// TIA Portal V17 export
// export: Created 2025-07-01T09:58:25.2131058Z, ExportSetting WithDefaults, DisplayName Totally Integrated Automation Portal, DisplayVersion V17 Update 8, DisplayName TIA Portal Openness, DisplayVersion V17 Update 8, DisplayName TIA Portal Version Control Interface, DisplayVersion V17, DisplayName SINAMICS Startdrive Advanced, DisplayVersion V17 SP2, DisplayName SINAMICS Startdrive G110M, G120, G120C, G120D, G120P, G115D, DisplayVersion V17 SP2, DisplayName SINAMICS Startdrive G130, G150, S120, S150, SINAMICS MV, S210, DisplayVersion V17 SP2, DisplayName STEP 7 Professional, DisplayVersion V17 Update 8, DisplayName SINUMERIK ONE STEP 7 Toolbox, DisplayVersion V17 Update 12, DisplayName SINUMERIK ONE PLC Basic Program Plus, DisplayVersion V17 Update 12, DisplayName SINUMERIK 840D sl STEP 7 Toolbox, DisplayVersion V17 Update 12, DisplayName STEP 7 Safety, DisplayVersion V17 Update 6, DisplayName WinCC Advanced, DisplayVersion V17 Update 8
FUNCTION "FC2441_MACHINE_STATUS" : Void   // FC2441, LAD
{ S7_Optimized_Access := 'TRUE' }
VERSION : 0.1
// stored: AutoNumber false, IsIECCheckEnabled false, SetENOAutomatically false, UDAEnableTagReadback false
BEGIN

REGION Network 1: UNIT 1 STATION 3 CLADDING IN PROCESS
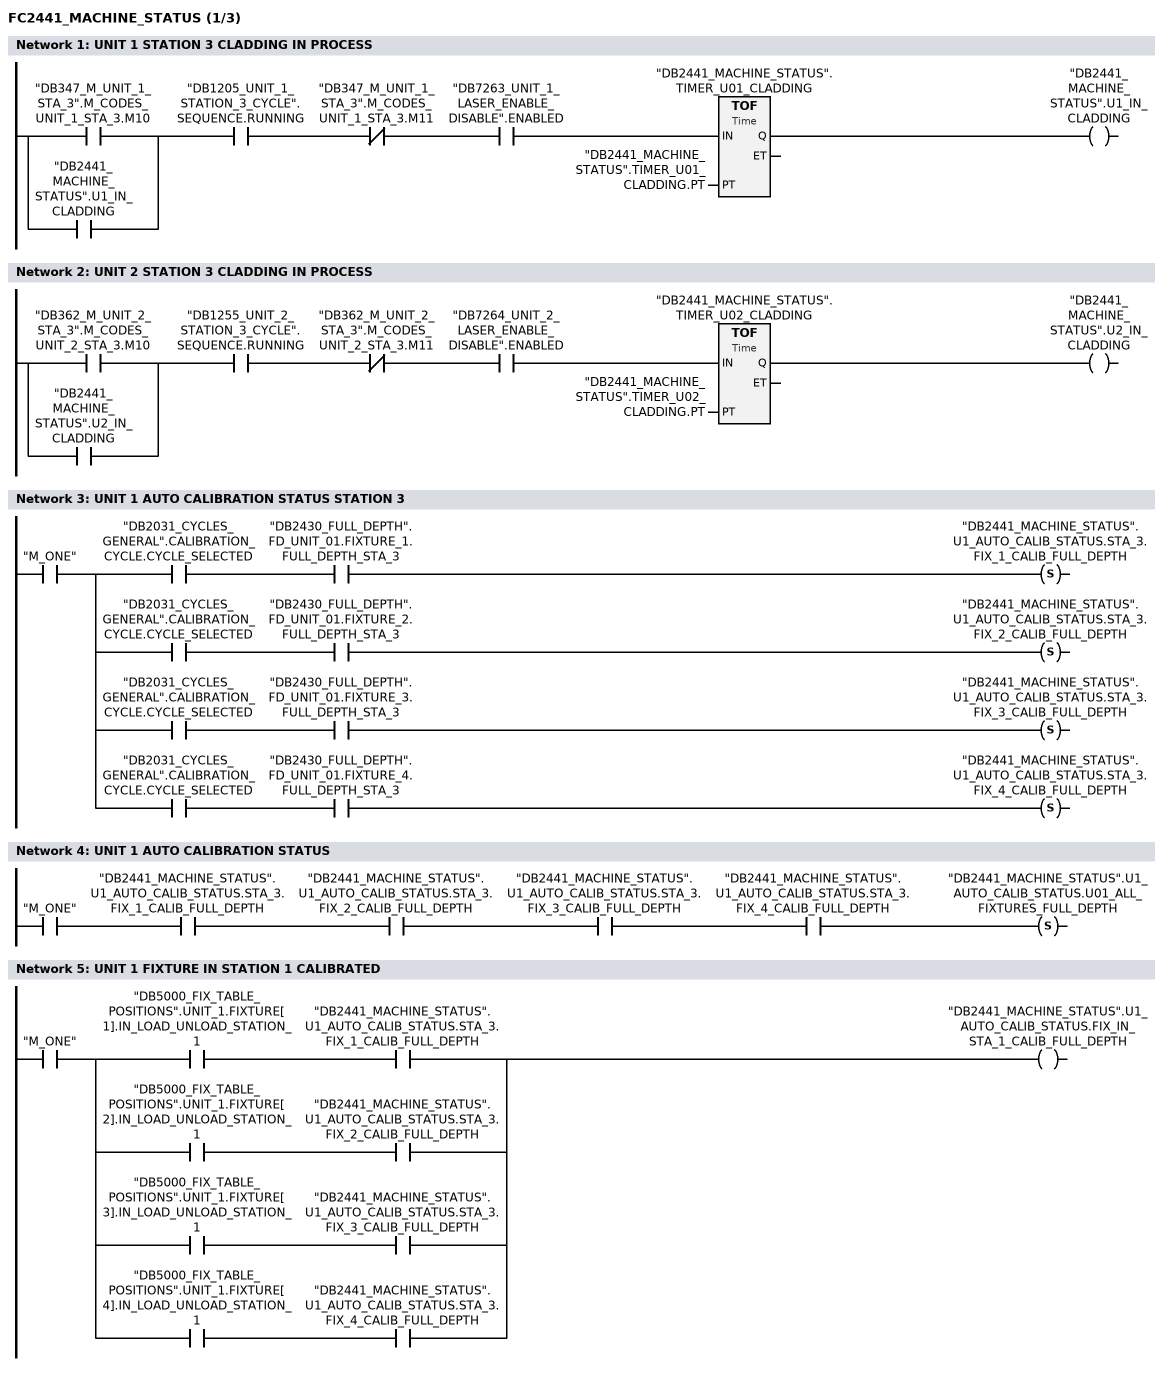
   RUNG wire#powerrail
      Contact( "DB347_M_UNIT_1_STA_3".M_CODES_UNIT_1_STA_3.M10 )
      wire#w1
      Contact( "DB1205_UNIT_1_STATION_3_CYCLE".SEQUENCE.RUNNING )
      I_Contact( "DB347_M_UNIT_1_STA_3".M_CODES_UNIT_1_STA_3.M11 )
      Contact( "DB7263_UNIT_1_LASER_ENABLE_DISABLE".ENABLED )
      { S7_Templates := "time_type := Time" } "DB2441_MACHINE_STATUS".TIMER_U01_CLADDING.TOF(pt := "DB2441_MACHINE_STATUS".TIMER_U01_CLADDING.PT, et =>)
      Coil( "DB2441_MACHINE_STATUS".U1_IN_CLADDING )
   END_RUNG
   RUNG wire#powerrail
      Contact( "DB2441_MACHINE_STATUS".U1_IN_CLADDING )
   END_RUNG wire#w1
   // the same network as SCL:
   "DB2441_MACHINE_STATUS".TIMER_U01_CLADDING.TOF(IN := ("DB347_M_UNIT_1_STA_3".M_CODES_UNIT_1_STA_3.M10 OR "DB2441_MACHINE_STATUS".U1_IN_CLADDING) AND "DB1205_UNIT_1_STATION_3_CYCLE".SEQUENCE.RUNNING AND NOT "DB347_M_UNIT_1_STA_3".M_CODES_UNIT_1_STA_3.M11 AND "DB7263_UNIT_1_LASER_ENABLE_DISABLE".ENABLED,
                           PT := "DB2441_MACHINE_STATUS".TIMER_U01_CLADDING.PT);
   "DB2441_MACHINE_STATUS".U1_IN_CLADDING := "DB2441_MACHINE_STATUS".TIMER_U01_CLADDING.Q;
END_REGION

REGION Network 2: UNIT 2 STATION 3 CLADDING IN PROCESS
   RUNG wire#powerrail
      Contact( "DB362_M_UNIT_2_STA_3".M_CODES_UNIT_2_STA_3.M10 )
      wire#w1
      Contact( "DB1255_UNIT_2_STATION_3_CYCLE".SEQUENCE.RUNNING )
      I_Contact( "DB362_M_UNIT_2_STA_3".M_CODES_UNIT_2_STA_3.M11 )
      Contact( "DB7264_UNIT_2_LASER_ENABLE_DISABLE".ENABLED )
      { S7_Templates := "time_type := Time" } "DB2441_MACHINE_STATUS".TIMER_U02_CLADDING.TOF(pt := "DB2441_MACHINE_STATUS".TIMER_U02_CLADDING.PT, et =>)
      Coil( "DB2441_MACHINE_STATUS".U2_IN_CLADDING )
   END_RUNG
   RUNG wire#powerrail
      Contact( "DB2441_MACHINE_STATUS".U2_IN_CLADDING )
   END_RUNG wire#w1
   // the same network as SCL:
   "DB2441_MACHINE_STATUS".TIMER_U02_CLADDING.TOF(IN := ("DB362_M_UNIT_2_STA_3".M_CODES_UNIT_2_STA_3.M10 OR "DB2441_MACHINE_STATUS".U2_IN_CLADDING) AND "DB1255_UNIT_2_STATION_3_CYCLE".SEQUENCE.RUNNING AND NOT "DB362_M_UNIT_2_STA_3".M_CODES_UNIT_2_STA_3.M11 AND "DB7264_UNIT_2_LASER_ENABLE_DISABLE".ENABLED,
                           PT := "DB2441_MACHINE_STATUS".TIMER_U02_CLADDING.PT);
   "DB2441_MACHINE_STATUS".U2_IN_CLADDING := "DB2441_MACHINE_STATUS".TIMER_U02_CLADDING.Q;
END_REGION

REGION Network 3: UNIT 1 AUTO CALIBRATION STATUS STATION 3
   RUNG wire#powerrail
      Contact( "M_ONE" )
      wire#w1
      Contact( "DB2031_CYCLES_GENERAL".CALIBRATION_CYCLE.CYCLE_SELECTED )
      Contact( "DB2430_FULL_DEPTH".FD_UNIT_01.FIXTURE_1.FULL_DEPTH_STA_3 )
      S_Coil( "DB2441_MACHINE_STATUS".U1_AUTO_CALIB_STATUS.STA_3.FIX_1_CALIB_FULL_DEPTH )
   END_RUNG
   RUNG wire#w1
      Contact( "DB2031_CYCLES_GENERAL".CALIBRATION_CYCLE.CYCLE_SELECTED )
      Contact( "DB2430_FULL_DEPTH".FD_UNIT_01.FIXTURE_2.FULL_DEPTH_STA_3 )
      S_Coil( "DB2441_MACHINE_STATUS".U1_AUTO_CALIB_STATUS.STA_3.FIX_2_CALIB_FULL_DEPTH )
   END_RUNG
   RUNG wire#w1
      Contact( "DB2031_CYCLES_GENERAL".CALIBRATION_CYCLE.CYCLE_SELECTED )
      Contact( "DB2430_FULL_DEPTH".FD_UNIT_01.FIXTURE_3.FULL_DEPTH_STA_3 )
      S_Coil( "DB2441_MACHINE_STATUS".U1_AUTO_CALIB_STATUS.STA_3.FIX_3_CALIB_FULL_DEPTH )
   END_RUNG
   RUNG wire#w1
      Contact( "DB2031_CYCLES_GENERAL".CALIBRATION_CYCLE.CYCLE_SELECTED )
      Contact( "DB2430_FULL_DEPTH".FD_UNIT_01.FIXTURE_4.FULL_DEPTH_STA_3 )
      S_Coil( "DB2441_MACHINE_STATUS".U1_AUTO_CALIB_STATUS.STA_3.FIX_4_CALIB_FULL_DEPTH )
   END_RUNG
   // the same network as SCL:
   IF "M_ONE" AND "DB2031_CYCLES_GENERAL".CALIBRATION_CYCLE.CYCLE_SELECTED AND "DB2430_FULL_DEPTH".FD_UNIT_01.FIXTURE_1.FULL_DEPTH_STA_3 THEN
       "DB2441_MACHINE_STATUS".U1_AUTO_CALIB_STATUS.STA_3.FIX_1_CALIB_FULL_DEPTH := TRUE;
   END_IF;
   IF "M_ONE" AND "DB2031_CYCLES_GENERAL".CALIBRATION_CYCLE.CYCLE_SELECTED AND "DB2430_FULL_DEPTH".FD_UNIT_01.FIXTURE_2.FULL_DEPTH_STA_3 THEN
       "DB2441_MACHINE_STATUS".U1_AUTO_CALIB_STATUS.STA_3.FIX_2_CALIB_FULL_DEPTH := TRUE;
   END_IF;
   IF "M_ONE" AND "DB2031_CYCLES_GENERAL".CALIBRATION_CYCLE.CYCLE_SELECTED AND "DB2430_FULL_DEPTH".FD_UNIT_01.FIXTURE_3.FULL_DEPTH_STA_3 THEN
       "DB2441_MACHINE_STATUS".U1_AUTO_CALIB_STATUS.STA_3.FIX_3_CALIB_FULL_DEPTH := TRUE;
   END_IF;
   IF "M_ONE" AND "DB2031_CYCLES_GENERAL".CALIBRATION_CYCLE.CYCLE_SELECTED AND "DB2430_FULL_DEPTH".FD_UNIT_01.FIXTURE_4.FULL_DEPTH_STA_3 THEN
       "DB2441_MACHINE_STATUS".U1_AUTO_CALIB_STATUS.STA_3.FIX_4_CALIB_FULL_DEPTH := TRUE;
   END_IF;
END_REGION

REGION Network 4: UNIT 1 AUTO CALIBRATION STATUS
   RUNG wire#powerrail
      Contact( "M_ONE" )
      Contact( "DB2441_MACHINE_STATUS".U1_AUTO_CALIB_STATUS.STA_3.FIX_1_CALIB_FULL_DEPTH )
      Contact( "DB2441_MACHINE_STATUS".U1_AUTO_CALIB_STATUS.STA_3.FIX_2_CALIB_FULL_DEPTH )
      Contact( "DB2441_MACHINE_STATUS".U1_AUTO_CALIB_STATUS.STA_3.FIX_3_CALIB_FULL_DEPTH )
      Contact( "DB2441_MACHINE_STATUS".U1_AUTO_CALIB_STATUS.STA_3.FIX_4_CALIB_FULL_DEPTH )
      S_Coil( "DB2441_MACHINE_STATUS".U1_AUTO_CALIB_STATUS.U01_ALL_FIXTURES_FULL_DEPTH )
   END_RUNG
   // the same network as SCL:
   IF "M_ONE" AND "DB2441_MACHINE_STATUS".U1_AUTO_CALIB_STATUS.STA_3.FIX_1_CALIB_FULL_DEPTH AND "DB2441_MACHINE_STATUS".U1_AUTO_CALIB_STATUS.STA_3.FIX_2_CALIB_FULL_DEPTH AND "DB2441_MACHINE_STATUS".U1_AUTO_CALIB_STATUS.STA_3.FIX_3_CALIB_FULL_DEPTH AND "DB2441_MACHINE_STATUS".U1_AUTO_CALIB_STATUS.STA_3.FIX_4_CALIB_FULL_DEPTH THEN
       "DB2441_MACHINE_STATUS".U1_AUTO_CALIB_STATUS.U01_ALL_FIXTURES_FULL_DEPTH := TRUE;
   END_IF;
END_REGION

REGION Network 5: UNIT 1 FIXTURE IN STATION 1 CALIBRATED
   RUNG wire#powerrail
      Contact( "M_ONE" )
      wire#w1
      Contact( "DB5000_FIX_TABLE_POSITIONS".UNIT_1.FIXTURE[1].IN_LOAD_UNLOAD_STATION_1 )
      Contact( "DB2441_MACHINE_STATUS".U1_AUTO_CALIB_STATUS.STA_3.FIX_1_CALIB_FULL_DEPTH )
      wire#w2
      Coil( "DB2441_MACHINE_STATUS".U1_AUTO_CALIB_STATUS.FIX_IN_STA_1_CALIB_FULL_DEPTH )
   END_RUNG
   RUNG wire#w1
      Contact( "DB5000_FIX_TABLE_POSITIONS".UNIT_1.FIXTURE[2].IN_LOAD_UNLOAD_STATION_1 )
      Contact( "DB2441_MACHINE_STATUS".U1_AUTO_CALIB_STATUS.STA_3.FIX_2_CALIB_FULL_DEPTH )
   END_RUNG wire#w2
   RUNG wire#w1
      Contact( "DB5000_FIX_TABLE_POSITIONS".UNIT_1.FIXTURE[3].IN_LOAD_UNLOAD_STATION_1 )
      Contact( "DB2441_MACHINE_STATUS".U1_AUTO_CALIB_STATUS.STA_3.FIX_3_CALIB_FULL_DEPTH )
   END_RUNG wire#w2
   RUNG wire#w1
      Contact( "DB5000_FIX_TABLE_POSITIONS".UNIT_1.FIXTURE[4].IN_LOAD_UNLOAD_STATION_1 )
      Contact( "DB2441_MACHINE_STATUS".U1_AUTO_CALIB_STATUS.STA_3.FIX_4_CALIB_FULL_DEPTH )
   END_RUNG wire#w2
   // the same network as SCL:
   "DB2441_MACHINE_STATUS".U1_AUTO_CALIB_STATUS.FIX_IN_STA_1_CALIB_FULL_DEPTH := "M_ONE" AND (("DB5000_FIX_TABLE_POSITIONS".UNIT_1.FIXTURE[1].IN_LOAD_UNLOAD_STATION_1 AND "DB2441_MACHINE_STATUS".U1_AUTO_CALIB_STATUS.STA_3.FIX_1_CALIB_FULL_DEPTH) OR ("DB5000_FIX_TABLE_POSITIONS".UNIT_1.FIXTURE[2].IN_LOAD_UNLOAD_STATION_1 AND "DB2441_MACHINE_STATUS".U1_AUTO_CALIB_STATUS.STA_3.FIX_2_CALIB_FULL_DEPTH) OR ("DB5000_FIX_TABLE_POSITIONS".UNIT_1.FIXTURE[3].IN_LOAD_UNLOAD_STATION_1 AND "DB2441_MACHINE_STATUS".U1_AUTO_CALIB_STATUS.STA_3.FIX_3_CALIB_FULL_DEPTH) OR ("DB5000_FIX_TABLE_POSITIONS".UNIT_1.FIXTURE[4].IN_LOAD_UNLOAD_STATION_1 AND "DB2441_MACHINE_STATUS".U1_AUTO_CALIB_STATUS.STA_3.FIX_4_CALIB_FULL_DEPTH));
END_REGION

REGION Network 6: UNIT 2 AUTO CALIBRATION STATUS STATION 2
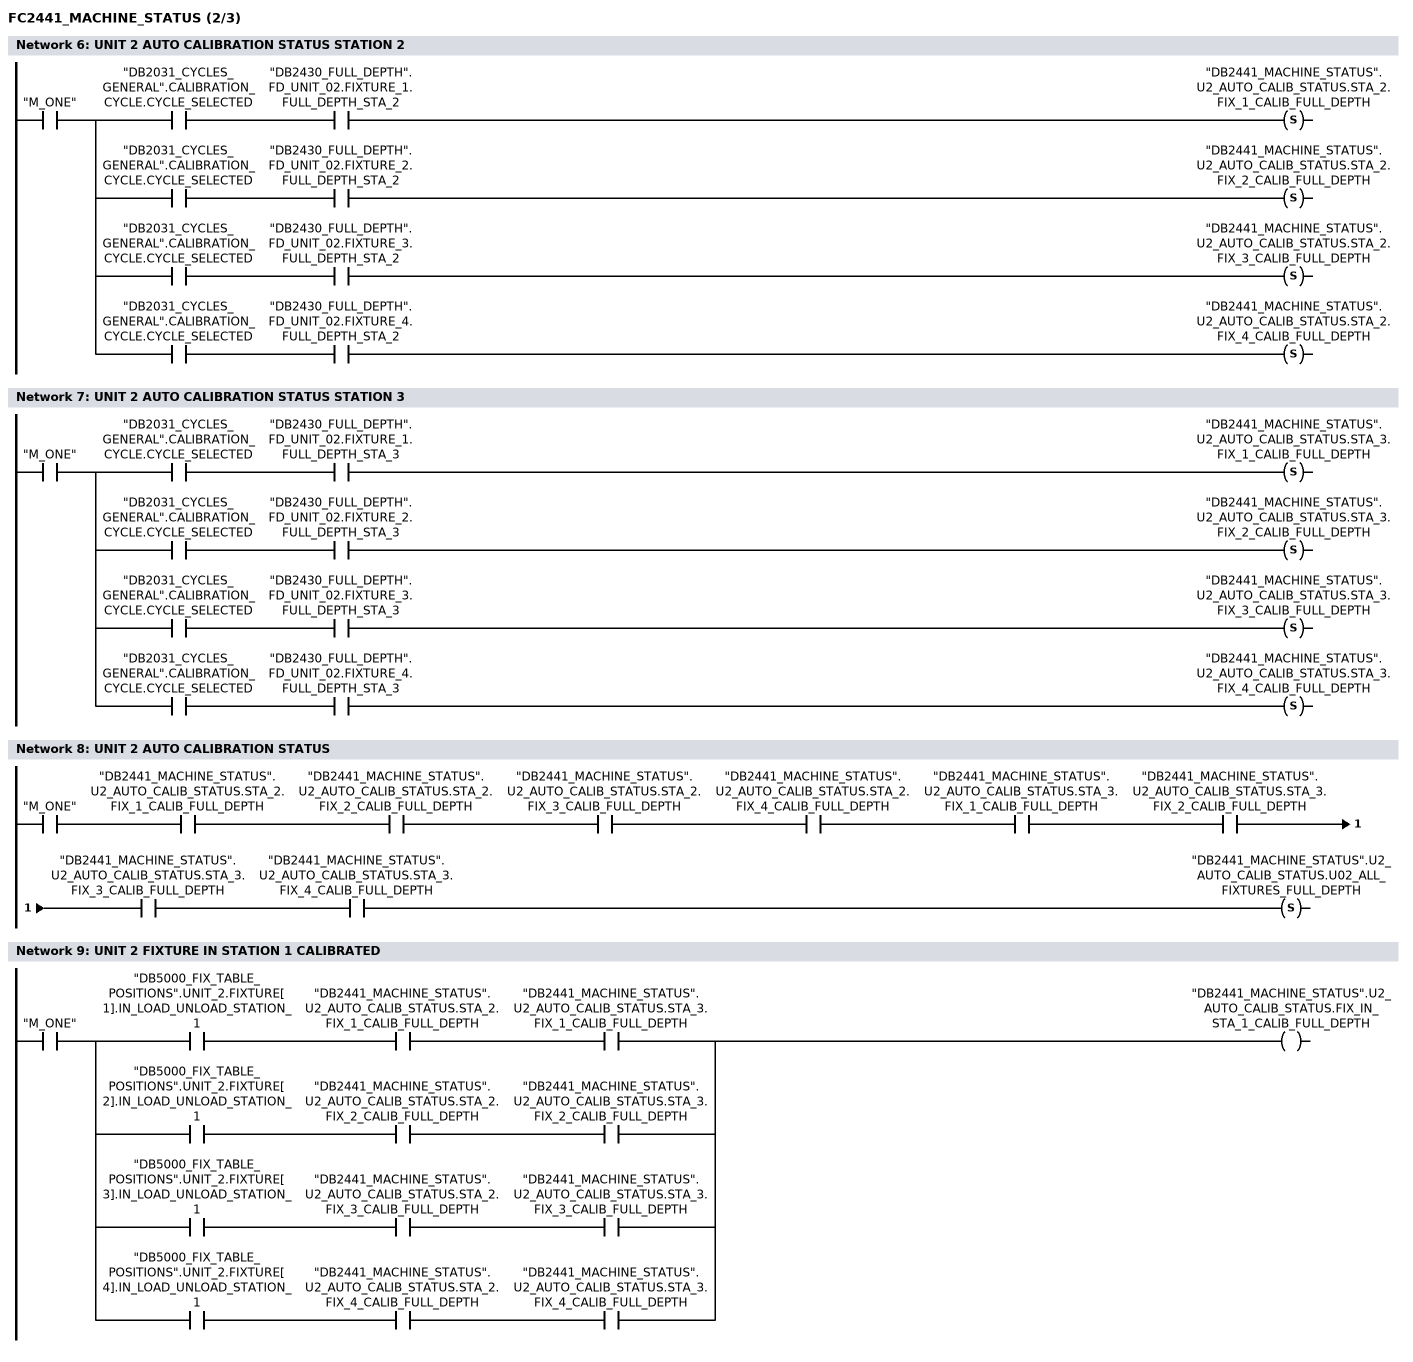
   RUNG wire#powerrail
      Contact( "M_ONE" )
      wire#w1
      Contact( "DB2031_CYCLES_GENERAL".CALIBRATION_CYCLE.CYCLE_SELECTED )
      Contact( "DB2430_FULL_DEPTH".FD_UNIT_02.FIXTURE_1.FULL_DEPTH_STA_2 )
      S_Coil( "DB2441_MACHINE_STATUS".U2_AUTO_CALIB_STATUS.STA_2.FIX_1_CALIB_FULL_DEPTH )
   END_RUNG
   RUNG wire#w1
      Contact( "DB2031_CYCLES_GENERAL".CALIBRATION_CYCLE.CYCLE_SELECTED )
      Contact( "DB2430_FULL_DEPTH".FD_UNIT_02.FIXTURE_2.FULL_DEPTH_STA_2 )
      S_Coil( "DB2441_MACHINE_STATUS".U2_AUTO_CALIB_STATUS.STA_2.FIX_2_CALIB_FULL_DEPTH )
   END_RUNG
   RUNG wire#w1
      Contact( "DB2031_CYCLES_GENERAL".CALIBRATION_CYCLE.CYCLE_SELECTED )
      Contact( "DB2430_FULL_DEPTH".FD_UNIT_02.FIXTURE_3.FULL_DEPTH_STA_2 )
      S_Coil( "DB2441_MACHINE_STATUS".U2_AUTO_CALIB_STATUS.STA_2.FIX_3_CALIB_FULL_DEPTH )
   END_RUNG
   RUNG wire#w1
      Contact( "DB2031_CYCLES_GENERAL".CALIBRATION_CYCLE.CYCLE_SELECTED )
      Contact( "DB2430_FULL_DEPTH".FD_UNIT_02.FIXTURE_4.FULL_DEPTH_STA_2 )
      S_Coil( "DB2441_MACHINE_STATUS".U2_AUTO_CALIB_STATUS.STA_2.FIX_4_CALIB_FULL_DEPTH )
   END_RUNG
   // the same network as SCL:
   IF "M_ONE" AND "DB2031_CYCLES_GENERAL".CALIBRATION_CYCLE.CYCLE_SELECTED AND "DB2430_FULL_DEPTH".FD_UNIT_02.FIXTURE_1.FULL_DEPTH_STA_2 THEN
       "DB2441_MACHINE_STATUS".U2_AUTO_CALIB_STATUS.STA_2.FIX_1_CALIB_FULL_DEPTH := TRUE;
   END_IF;
   IF "M_ONE" AND "DB2031_CYCLES_GENERAL".CALIBRATION_CYCLE.CYCLE_SELECTED AND "DB2430_FULL_DEPTH".FD_UNIT_02.FIXTURE_2.FULL_DEPTH_STA_2 THEN
       "DB2441_MACHINE_STATUS".U2_AUTO_CALIB_STATUS.STA_2.FIX_2_CALIB_FULL_DEPTH := TRUE;
   END_IF;
   IF "M_ONE" AND "DB2031_CYCLES_GENERAL".CALIBRATION_CYCLE.CYCLE_SELECTED AND "DB2430_FULL_DEPTH".FD_UNIT_02.FIXTURE_3.FULL_DEPTH_STA_2 THEN
       "DB2441_MACHINE_STATUS".U2_AUTO_CALIB_STATUS.STA_2.FIX_3_CALIB_FULL_DEPTH := TRUE;
   END_IF;
   IF "M_ONE" AND "DB2031_CYCLES_GENERAL".CALIBRATION_CYCLE.CYCLE_SELECTED AND "DB2430_FULL_DEPTH".FD_UNIT_02.FIXTURE_4.FULL_DEPTH_STA_2 THEN
       "DB2441_MACHINE_STATUS".U2_AUTO_CALIB_STATUS.STA_2.FIX_4_CALIB_FULL_DEPTH := TRUE;
   END_IF;
END_REGION

REGION Network 7: UNIT 2 AUTO CALIBRATION STATUS STATION 3
   RUNG wire#powerrail
      Contact( "M_ONE" )
      wire#w1
      Contact( "DB2031_CYCLES_GENERAL".CALIBRATION_CYCLE.CYCLE_SELECTED )
      Contact( "DB2430_FULL_DEPTH".FD_UNIT_02.FIXTURE_1.FULL_DEPTH_STA_3 )
      S_Coil( "DB2441_MACHINE_STATUS".U2_AUTO_CALIB_STATUS.STA_3.FIX_1_CALIB_FULL_DEPTH )
   END_RUNG
   RUNG wire#w1
      Contact( "DB2031_CYCLES_GENERAL".CALIBRATION_CYCLE.CYCLE_SELECTED )
      Contact( "DB2430_FULL_DEPTH".FD_UNIT_02.FIXTURE_2.FULL_DEPTH_STA_3 )
      S_Coil( "DB2441_MACHINE_STATUS".U2_AUTO_CALIB_STATUS.STA_3.FIX_2_CALIB_FULL_DEPTH )
   END_RUNG
   RUNG wire#w1
      Contact( "DB2031_CYCLES_GENERAL".CALIBRATION_CYCLE.CYCLE_SELECTED )
      Contact( "DB2430_FULL_DEPTH".FD_UNIT_02.FIXTURE_3.FULL_DEPTH_STA_3 )
      S_Coil( "DB2441_MACHINE_STATUS".U2_AUTO_CALIB_STATUS.STA_3.FIX_3_CALIB_FULL_DEPTH )
   END_RUNG
   RUNG wire#w1
      Contact( "DB2031_CYCLES_GENERAL".CALIBRATION_CYCLE.CYCLE_SELECTED )
      Contact( "DB2430_FULL_DEPTH".FD_UNIT_02.FIXTURE_4.FULL_DEPTH_STA_3 )
      S_Coil( "DB2441_MACHINE_STATUS".U2_AUTO_CALIB_STATUS.STA_3.FIX_4_CALIB_FULL_DEPTH )
   END_RUNG
   // the same network as SCL:
   IF "M_ONE" AND "DB2031_CYCLES_GENERAL".CALIBRATION_CYCLE.CYCLE_SELECTED AND "DB2430_FULL_DEPTH".FD_UNIT_02.FIXTURE_1.FULL_DEPTH_STA_3 THEN
       "DB2441_MACHINE_STATUS".U2_AUTO_CALIB_STATUS.STA_3.FIX_1_CALIB_FULL_DEPTH := TRUE;
   END_IF;
   IF "M_ONE" AND "DB2031_CYCLES_GENERAL".CALIBRATION_CYCLE.CYCLE_SELECTED AND "DB2430_FULL_DEPTH".FD_UNIT_02.FIXTURE_2.FULL_DEPTH_STA_3 THEN
       "DB2441_MACHINE_STATUS".U2_AUTO_CALIB_STATUS.STA_3.FIX_2_CALIB_FULL_DEPTH := TRUE;
   END_IF;
   IF "M_ONE" AND "DB2031_CYCLES_GENERAL".CALIBRATION_CYCLE.CYCLE_SELECTED AND "DB2430_FULL_DEPTH".FD_UNIT_02.FIXTURE_3.FULL_DEPTH_STA_3 THEN
       "DB2441_MACHINE_STATUS".U2_AUTO_CALIB_STATUS.STA_3.FIX_3_CALIB_FULL_DEPTH := TRUE;
   END_IF;
   IF "M_ONE" AND "DB2031_CYCLES_GENERAL".CALIBRATION_CYCLE.CYCLE_SELECTED AND "DB2430_FULL_DEPTH".FD_UNIT_02.FIXTURE_4.FULL_DEPTH_STA_3 THEN
       "DB2441_MACHINE_STATUS".U2_AUTO_CALIB_STATUS.STA_3.FIX_4_CALIB_FULL_DEPTH := TRUE;
   END_IF;
END_REGION

REGION Network 8: UNIT 2 AUTO CALIBRATION STATUS
   RUNG wire#powerrail
      Contact( "M_ONE" )
      Contact( "DB2441_MACHINE_STATUS".U2_AUTO_CALIB_STATUS.STA_2.FIX_1_CALIB_FULL_DEPTH )
      Contact( "DB2441_MACHINE_STATUS".U2_AUTO_CALIB_STATUS.STA_2.FIX_2_CALIB_FULL_DEPTH )
      Contact( "DB2441_MACHINE_STATUS".U2_AUTO_CALIB_STATUS.STA_2.FIX_3_CALIB_FULL_DEPTH )
      Contact( "DB2441_MACHINE_STATUS".U2_AUTO_CALIB_STATUS.STA_2.FIX_4_CALIB_FULL_DEPTH )
      Contact( "DB2441_MACHINE_STATUS".U2_AUTO_CALIB_STATUS.STA_3.FIX_1_CALIB_FULL_DEPTH )
      Contact( "DB2441_MACHINE_STATUS".U2_AUTO_CALIB_STATUS.STA_3.FIX_2_CALIB_FULL_DEPTH )
      Contact( "DB2441_MACHINE_STATUS".U2_AUTO_CALIB_STATUS.STA_3.FIX_3_CALIB_FULL_DEPTH )
      Contact( "DB2441_MACHINE_STATUS".U2_AUTO_CALIB_STATUS.STA_3.FIX_4_CALIB_FULL_DEPTH )
      S_Coil( "DB2441_MACHINE_STATUS".U2_AUTO_CALIB_STATUS.U02_ALL_FIXTURES_FULL_DEPTH )
   END_RUNG
   // the same network as SCL:
   IF "M_ONE" AND "DB2441_MACHINE_STATUS".U2_AUTO_CALIB_STATUS.STA_2.FIX_1_CALIB_FULL_DEPTH AND "DB2441_MACHINE_STATUS".U2_AUTO_CALIB_STATUS.STA_2.FIX_2_CALIB_FULL_DEPTH AND "DB2441_MACHINE_STATUS".U2_AUTO_CALIB_STATUS.STA_2.FIX_3_CALIB_FULL_DEPTH AND "DB2441_MACHINE_STATUS".U2_AUTO_CALIB_STATUS.STA_2.FIX_4_CALIB_FULL_DEPTH AND "DB2441_MACHINE_STATUS".U2_AUTO_CALIB_STATUS.STA_3.FIX_1_CALIB_FULL_DEPTH AND "DB2441_MACHINE_STATUS".U2_AUTO_CALIB_STATUS.STA_3.FIX_2_CALIB_FULL_DEPTH AND "DB2441_MACHINE_STATUS".U2_AUTO_CALIB_STATUS.STA_3.FIX_3_CALIB_FULL_DEPTH AND "DB2441_MACHINE_STATUS".U2_AUTO_CALIB_STATUS.STA_3.FIX_4_CALIB_FULL_DEPTH THEN
       "DB2441_MACHINE_STATUS".U2_AUTO_CALIB_STATUS.U02_ALL_FIXTURES_FULL_DEPTH := TRUE;
   END_IF;
END_REGION

REGION Network 9: UNIT 2 FIXTURE IN STATION 1 CALIBRATED
   RUNG wire#powerrail
      Contact( "M_ONE" )
      wire#w1
      Contact( "DB5000_FIX_TABLE_POSITIONS".UNIT_2.FIXTURE[1].IN_LOAD_UNLOAD_STATION_1 )
      Contact( "DB2441_MACHINE_STATUS".U2_AUTO_CALIB_STATUS.STA_2.FIX_1_CALIB_FULL_DEPTH )
      Contact( "DB2441_MACHINE_STATUS".U2_AUTO_CALIB_STATUS.STA_3.FIX_1_CALIB_FULL_DEPTH )
      wire#w2
      Coil( "DB2441_MACHINE_STATUS".U2_AUTO_CALIB_STATUS.FIX_IN_STA_1_CALIB_FULL_DEPTH )
   END_RUNG
   RUNG wire#w1
      Contact( "DB5000_FIX_TABLE_POSITIONS".UNIT_2.FIXTURE[2].IN_LOAD_UNLOAD_STATION_1 )
      Contact( "DB2441_MACHINE_STATUS".U2_AUTO_CALIB_STATUS.STA_2.FIX_2_CALIB_FULL_DEPTH )
      Contact( "DB2441_MACHINE_STATUS".U2_AUTO_CALIB_STATUS.STA_3.FIX_2_CALIB_FULL_DEPTH )
   END_RUNG wire#w2
   RUNG wire#w1
      Contact( "DB5000_FIX_TABLE_POSITIONS".UNIT_2.FIXTURE[3].IN_LOAD_UNLOAD_STATION_1 )
      Contact( "DB2441_MACHINE_STATUS".U2_AUTO_CALIB_STATUS.STA_2.FIX_3_CALIB_FULL_DEPTH )
      Contact( "DB2441_MACHINE_STATUS".U2_AUTO_CALIB_STATUS.STA_3.FIX_3_CALIB_FULL_DEPTH )
   END_RUNG wire#w2
   RUNG wire#w1
      Contact( "DB5000_FIX_TABLE_POSITIONS".UNIT_2.FIXTURE[4].IN_LOAD_UNLOAD_STATION_1 )
      Contact( "DB2441_MACHINE_STATUS".U2_AUTO_CALIB_STATUS.STA_2.FIX_4_CALIB_FULL_DEPTH )
      Contact( "DB2441_MACHINE_STATUS".U2_AUTO_CALIB_STATUS.STA_3.FIX_4_CALIB_FULL_DEPTH )
   END_RUNG wire#w2
   // the same network as SCL:
   "DB2441_MACHINE_STATUS".U2_AUTO_CALIB_STATUS.FIX_IN_STA_1_CALIB_FULL_DEPTH := "M_ONE" AND (("DB5000_FIX_TABLE_POSITIONS".UNIT_2.FIXTURE[1].IN_LOAD_UNLOAD_STATION_1 AND "DB2441_MACHINE_STATUS".U2_AUTO_CALIB_STATUS.STA_2.FIX_1_CALIB_FULL_DEPTH AND "DB2441_MACHINE_STATUS".U2_AUTO_CALIB_STATUS.STA_3.FIX_1_CALIB_FULL_DEPTH) OR ("DB5000_FIX_TABLE_POSITIONS".UNIT_2.FIXTURE[2].IN_LOAD_UNLOAD_STATION_1 AND "DB2441_MACHINE_STATUS".U2_AUTO_CALIB_STATUS.STA_2.FIX_2_CALIB_FULL_DEPTH AND "DB2441_MACHINE_STATUS".U2_AUTO_CALIB_STATUS.STA_3.FIX_2_CALIB_FULL_DEPTH) OR ("DB5000_FIX_TABLE_POSITIONS".UNIT_2.FIXTURE[3].IN_LOAD_UNLOAD_STATION_1 AND "DB2441_MACHINE_STATUS".U2_AUTO_CALIB_STATUS.STA_2.FIX_3_CALIB_FULL_DEPTH AND "DB2441_MACHINE_STATUS".U2_AUTO_CALIB_STATUS.STA_3.FIX_3_CALIB_FULL_DEPTH) OR ("DB5000_FIX_TABLE_POSITIONS".UNIT_2.FIXTURE[4].IN_LOAD_UNLOAD_STATION_1 AND "DB2441_MACHINE_STATUS".U2_AUTO_CALIB_STATUS.STA_2.FIX_4_CALIB_FULL_DEPTH AND "DB2441_MACHINE_STATUS".U2_AUTO_CALIB_STATUS.STA_3.FIX_4_CALIB_FULL_DEPTH));
END_REGION

REGION Network 10: UNIT 3 AUTO CALIBRATION STATUS
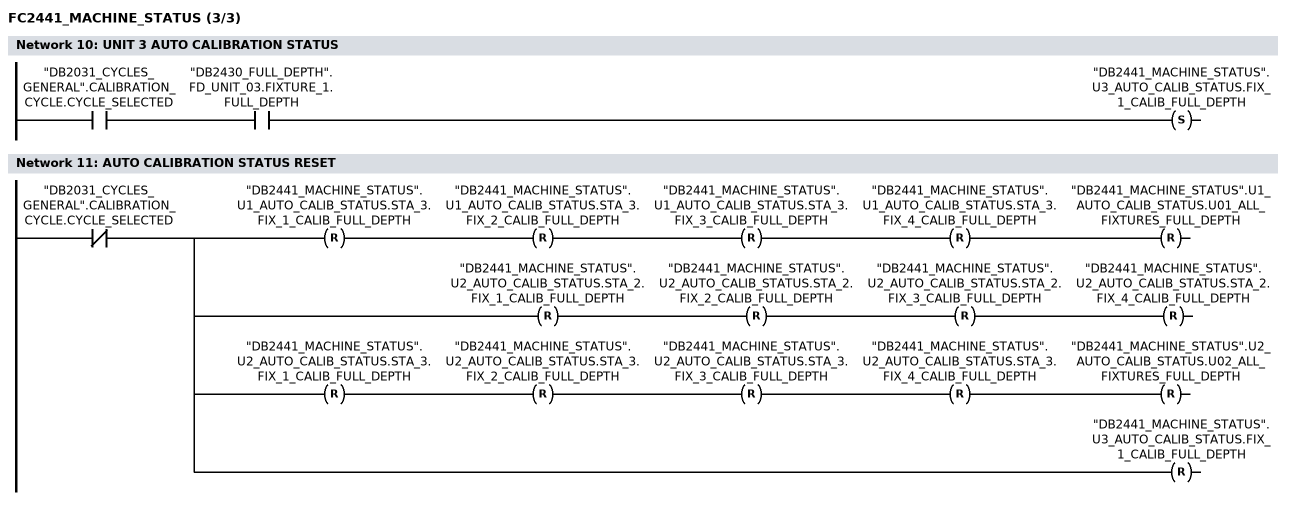
   RUNG wire#powerrail
      Contact( "DB2031_CYCLES_GENERAL".CALIBRATION_CYCLE.CYCLE_SELECTED )
      Contact( "DB2430_FULL_DEPTH".FD_UNIT_03.FIXTURE_1.FULL_DEPTH )
      S_Coil( "DB2441_MACHINE_STATUS".U3_AUTO_CALIB_STATUS.FIX_1_CALIB_FULL_DEPTH )
   END_RUNG
   // the same network as SCL:
   IF "DB2031_CYCLES_GENERAL".CALIBRATION_CYCLE.CYCLE_SELECTED AND "DB2430_FULL_DEPTH".FD_UNIT_03.FIXTURE_1.FULL_DEPTH THEN
       "DB2441_MACHINE_STATUS".U3_AUTO_CALIB_STATUS.FIX_1_CALIB_FULL_DEPTH := TRUE;
   END_IF;
END_REGION

REGION Network 11: AUTO CALIBRATION STATUS RESET
   RUNG wire#powerrail
      I_Contact( "DB2031_CYCLES_GENERAL".CALIBRATION_CYCLE.CYCLE_SELECTED )
      wire#w1
      R_Coil( "DB2441_MACHINE_STATUS".U1_AUTO_CALIB_STATUS.STA_3.FIX_1_CALIB_FULL_DEPTH )
      R_Coil( "DB2441_MACHINE_STATUS".U1_AUTO_CALIB_STATUS.STA_3.FIX_2_CALIB_FULL_DEPTH )
      R_Coil( "DB2441_MACHINE_STATUS".U1_AUTO_CALIB_STATUS.STA_3.FIX_3_CALIB_FULL_DEPTH )
      R_Coil( "DB2441_MACHINE_STATUS".U1_AUTO_CALIB_STATUS.STA_3.FIX_4_CALIB_FULL_DEPTH )
      R_Coil( "DB2441_MACHINE_STATUS".U1_AUTO_CALIB_STATUS.U01_ALL_FIXTURES_FULL_DEPTH )
   END_RUNG
   RUNG wire#w1
      R_Coil( "DB2441_MACHINE_STATUS".U2_AUTO_CALIB_STATUS.STA_2.FIX_1_CALIB_FULL_DEPTH )
      R_Coil( "DB2441_MACHINE_STATUS".U2_AUTO_CALIB_STATUS.STA_2.FIX_2_CALIB_FULL_DEPTH )
      R_Coil( "DB2441_MACHINE_STATUS".U2_AUTO_CALIB_STATUS.STA_2.FIX_3_CALIB_FULL_DEPTH )
      R_Coil( "DB2441_MACHINE_STATUS".U2_AUTO_CALIB_STATUS.STA_2.FIX_4_CALIB_FULL_DEPTH )
   END_RUNG
   RUNG wire#w1
      R_Coil( "DB2441_MACHINE_STATUS".U2_AUTO_CALIB_STATUS.STA_3.FIX_1_CALIB_FULL_DEPTH )
      R_Coil( "DB2441_MACHINE_STATUS".U2_AUTO_CALIB_STATUS.STA_3.FIX_2_CALIB_FULL_DEPTH )
      R_Coil( "DB2441_MACHINE_STATUS".U2_AUTO_CALIB_STATUS.STA_3.FIX_3_CALIB_FULL_DEPTH )
      R_Coil( "DB2441_MACHINE_STATUS".U2_AUTO_CALIB_STATUS.STA_3.FIX_4_CALIB_FULL_DEPTH )
      R_Coil( "DB2441_MACHINE_STATUS".U2_AUTO_CALIB_STATUS.U02_ALL_FIXTURES_FULL_DEPTH )
   END_RUNG
   RUNG wire#w1
      R_Coil( "DB2441_MACHINE_STATUS".U3_AUTO_CALIB_STATUS.FIX_1_CALIB_FULL_DEPTH )
   END_RUNG
   // the same network as SCL:
   IF NOT "DB2031_CYCLES_GENERAL".CALIBRATION_CYCLE.CYCLE_SELECTED THEN
       "DB2441_MACHINE_STATUS".U1_AUTO_CALIB_STATUS.STA_3.FIX_1_CALIB_FULL_DEPTH := FALSE;
       "DB2441_MACHINE_STATUS".U1_AUTO_CALIB_STATUS.STA_3.FIX_2_CALIB_FULL_DEPTH := FALSE;
       "DB2441_MACHINE_STATUS".U1_AUTO_CALIB_STATUS.STA_3.FIX_3_CALIB_FULL_DEPTH := FALSE;
       "DB2441_MACHINE_STATUS".U1_AUTO_CALIB_STATUS.STA_3.FIX_4_CALIB_FULL_DEPTH := FALSE;
       "DB2441_MACHINE_STATUS".U1_AUTO_CALIB_STATUS.U01_ALL_FIXTURES_FULL_DEPTH := FALSE;
       "DB2441_MACHINE_STATUS".U2_AUTO_CALIB_STATUS.STA_2.FIX_1_CALIB_FULL_DEPTH := FALSE;
       "DB2441_MACHINE_STATUS".U2_AUTO_CALIB_STATUS.STA_2.FIX_2_CALIB_FULL_DEPTH := FALSE;
       "DB2441_MACHINE_STATUS".U2_AUTO_CALIB_STATUS.STA_2.FIX_3_CALIB_FULL_DEPTH := FALSE;
       "DB2441_MACHINE_STATUS".U2_AUTO_CALIB_STATUS.STA_2.FIX_4_CALIB_FULL_DEPTH := FALSE;
       "DB2441_MACHINE_STATUS".U2_AUTO_CALIB_STATUS.STA_3.FIX_1_CALIB_FULL_DEPTH := FALSE;
       "DB2441_MACHINE_STATUS".U2_AUTO_CALIB_STATUS.STA_3.FIX_2_CALIB_FULL_DEPTH := FALSE;
       "DB2441_MACHINE_STATUS".U2_AUTO_CALIB_STATUS.STA_3.FIX_3_CALIB_FULL_DEPTH := FALSE;
       "DB2441_MACHINE_STATUS".U2_AUTO_CALIB_STATUS.STA_3.FIX_4_CALIB_FULL_DEPTH := FALSE;
       "DB2441_MACHINE_STATUS".U2_AUTO_CALIB_STATUS.U02_ALL_FIXTURES_FULL_DEPTH := FALSE;
       "DB2441_MACHINE_STATUS".U3_AUTO_CALIB_STATUS.FIX_1_CALIB_FULL_DEPTH := FALSE;
   END_IF;
END_REGION
END_FUNCTION
